{attribute addProperty BoxType "EL3423-0000-0016"}
{attribute addProperty Id "TxPDO_ToggleAT %I*BOOL8116Active_EnergyAT %I*REAL32417Active_Energy_PositiveAT %I*REAL32418Active_Energy_NegativeAT %I*REAL32419Apparent_EnergyAT %I*REAL32420Apparent_Energy_PositiveAT %I*REAL32421Apparent_Energy_NegativeAT %I*REAL32422Reactive_EnergyAT %I*REAL32423Reactive_Energy_PositiveAT %I*REAL32424Reactive_Energy_NegativeAT %I*REAL32425"}
{attribute addProperty CRC "998821580"}
{attribute addProperty SizeInBites "296"}
{attribute addProperty SizeInBytes "37"}
TYPE Total_Interval_Energy_3B88CECC :
STRUCT
	{attribute addProperty Name "TxPDO_Toggle"}
	TxPDO_Toggle AT %I* : BOOL;
	{attribute addProperty Name "Active_Energy"}
	Active_Energy AT %I* : REAL;
	{attribute addProperty Name "Active_Energy_Positive"}
	Active_Energy_Positive AT %I* : REAL;
	{attribute addProperty Name "Active_Energy_Negative"}
	Active_Energy_Negative AT %I* : REAL;
	{attribute addProperty Name "Apparent_Energy"}
	Apparent_Energy AT %I* : REAL;
	{attribute addProperty Name "Apparent_Energy_Positive"}
	Apparent_Energy_Positive AT %I* : REAL;
	{attribute addProperty Name "Apparent_Energy_Negative"}
	Apparent_Energy_Negative AT %I* : REAL;
	{attribute addProperty Name "Reactive_Energy"}
	Reactive_Energy AT %I* : REAL;
	{attribute addProperty Name "Reactive_Energy_Positive"}
	Reactive_Energy_Positive AT %I* : REAL;
	{attribute addProperty Name "Reactive_Energy_Negative"}
	Reactive_Energy_Negative AT %I* : REAL;
END_STRUCT
END_TYPE

(* stored: Version 1.2.0.0, ProductVersion 3.1.4024.9
   DUT Total_Interval_Energy_3B88CECC: Id {98a95ffd-d090-4694-9218-8cd772630d60} *)
